// TwinCAT 3 PLC project main
// ProgramVersion: 3.1.4024.0
// libraries:
//   Tc2_Standard, * (Beckhoff Automation GmbH)
//   Tc2_System, * (Beckhoff Automation GmbH)
//   Tc3_Module, * (Beckhoff Automation GmbH)
// project tree:
//   / GlobalTextList.TcGTLO, PlcTask.TcTTO, Visualization Manager.TcVMO (not stored)
//   POUs/ MAIN.TcPOU
//   VISUs/ Visu.TcVIS
// real-time tasks:
//   TASK PlcTask: cycle T#10ms, priority 20, ADS port 350

CONFIGURATION main
    RESOURCE PLC ON TwinCAT3
        TASK PlcTask(INTERVAL := T#10ms, PRIORITY := 20);
        PROGRAM MAIN WITH PlcTask : MAIN;
    END_RESOURCE
END_CONFIGURATION

// ---- POUs/MAIN.TcPOU
PROGRAM MAIN
VAR
	nVat1 : INT; //Niveau vat 1
	nVat2 : INT; //Niveau vat 2
	nVat3 : INT; //Niveau vat 3
	
	nTotaal : int; //Totaal van alle vaten
END_VAR

//De inhoud van 3 vaten wordt afzonderlijk gemeten en kunnen maximaal 2000L, 3000L en 5000L bevatten.
//De waarde die men inleest is de hoeveelheid die zich in het vat bevindt (nVat1, nVat2 en nVat3). 

//Simuleer deze ingangen. Bouw een visualisatie die de inhoud van elke tank afzonderlijk alsook de som weergeeft.
//Maak gebruik van 3 sliders en 1 bar display. Houd eveneens rekening met de maximum waarden.

nTotaal := nVat1 + nVat2 + nVat3;

END_PROGRAM

// ---- GlobalTextList.TcGTLO
TEXTLIST GlobalTextList
  56 = 'Label'
  302 = 'nVat1'
  571 = 'nVat2'
  179 = 'nVat3'
END_TEXTLIST

// ---- VISUs/Visu.TcVIS
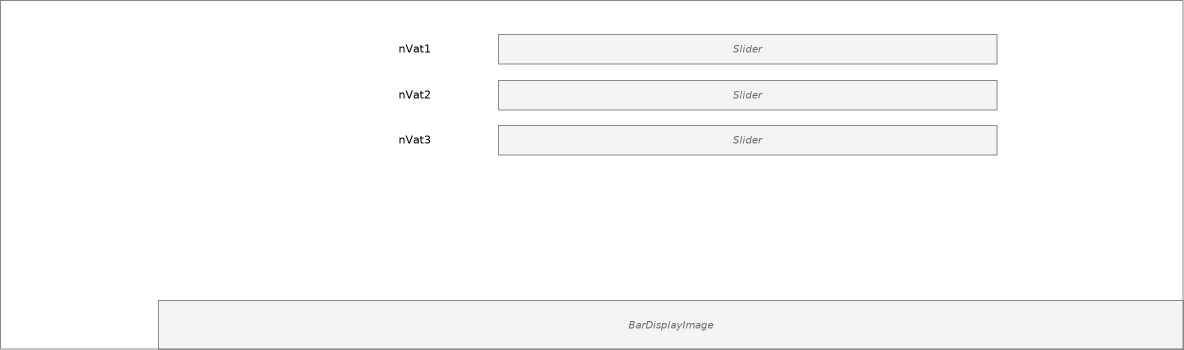
VISUALIZATION Visu  // 1184x350
    Slider (498,34 499x30), variable: MAIN.nVat1, scale 0..2000
    Slider (498,80 499x30), variable: MAIN.nVat2, scale 0..3000
    Slider (498,125 499x30), variable: MAIN.nVat3, scale 0..5000
    Label (340,34 150x30), "nVat1"
    Label (340,80 150x30), "nVat2"
    Label (340,125 150x30), "nVat3"
    BarDisplayImage (158,300 1026x50), value: MAIN.nTotaal, style: BarDisplayImage-Gray, scale format: %.1f, scale 0..10000
END_VISUALIZATION
